PROGRAM prgWeatherStations
VAR
	{attribute wpf [Container(Layout.Wrap)]}
	_weatherStationsCyclicAccess : fbWorldWeatherWatch;
	_weatherStationsBatchAccess : fbWorldWeatherWatch;
	_weatherStationsSynchronAccess : fbWorldWeatherWatch;
END_VAR

_weatherStationsCyclicAccess();
_weatherStationsBatchAccess();
_weatherStationsSynchronAccess();

END_PROGRAM

(* stored: Version 1.1.0.1, ProductVersion 3.1.4024.0
   POU prgWeatherStations: Id {63837f3c-745d-4340-ad1b-7cd9b6b37ded}, SpecialFunc None *)
